{region '#Template'}
	{attribute 'Version' := '5.0.0.0'}
	{attribute 'Tags' := '"LCID": "1031", "Text": "Trade, Plant, Room automation"'}
	{attribute 'Tags' := '"LCID": "1033", "Text": "Trade, Plant, Room automation"'}
	{attribute 'Using' := '"Type": "Template", "URI": "Site"'}
	{attribute 'Description' := '"LCID": "1031", "Text": "Aufruf der Anlagen des Gewerks Raumautomation"'}
	{attribute 'Description' := '"LCID": "1033", "Text": "Calling the plants of the trade room automation"'}
{endregion}
FUNCTION_BLOCK FB_BA_RoomAutomationServer EXTENDS FB_BA_View
VAR_INPUT CONSTANT
	AdsComServerRoom	: FB_BA_AdsComServer_Room;
	BuildingData		: FB_BA_BuildingData;
	
	RoomSample			: FB_BA_RoomSample1;
END_VAR

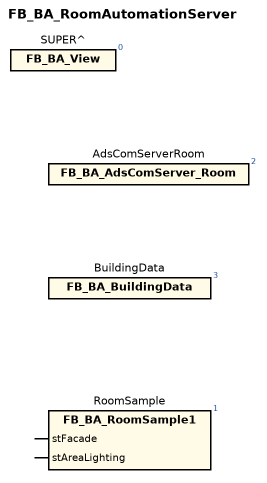
SUPER^(); // FB_BA_View
RoomSample(); // FB_BA_RoomSample1
AdsComServerRoom(); // FB_BA_AdsComServer_Room
BuildingData(); // FB_BA_BuildingData

METHOD FB_init : BOOL
VAR_INPUT
	bInitRetains : BOOL; // if TRUE, the retain variables are initialized (warm start / cold start)
	bInCopyCode : BOOL;  // if TRUE, the instance afterwards gets moved into the copy code (online change)
END_VAR
BuildingData.iParent			:= THIS^;	
BuildingData.iLabel				:= LblPlt_Global_building_data;
BuildingData.sObjectName		:= '{Idx=01}';
BuildingData.eDPADMode			:= E_BA_DPADMode.eInclude;

RoomSample.iParent 				:= THIS^;	
RoomSample.sObjectName			:= '{ROM}';	
RoomSample.sDescription			:= '{Room 01}';  
RoomSample.eDPADMode			:= E_BA_DPADMode.eInclude;
END_METHOD

END_FUNCTION_BLOCK

(* stored: Version 1.1.0.1, ProductVersion 3.1.4024.13
   POU FB_BA_RoomAutomationServer: Id {8aa4396b-0cd5-4ea5-b2b2-02d92281492e}, SpecialFunc None
   Method FB_init: Id {4b1b0a6f-5200-4809-af0e-3278ef788af7} *)
